# B&R Automation Studio project Cognex_V1_5
Automation Studio 4.6.3.55

## Configuration PP500_15

CPU , AutomationRuntime B4.62, Build 4.1.2, Safety 1.6, Vc V4.62.0

### Task classes (Cpu.sw)
```
Cyclic#8 (cycle 4000 us):
  Cognex <- Cognex.prg
  CognexVisN <- CognexVisNativeMode.prg
  CognexVisC <- CognexVisCommissioning.prg
  CognexVisA <- CognexVisArchive.prg
  CognexVisM <- CognexVisMain.prg
VcDataObjects: Visu <- Visu.dob, Visu1 <- Visu.dob
Binaries: vcclbox, vcctext, vcrt, vcresman, vccbar, vccstr, vccurl, vcchtml, vcpfmtcx, vcptelo, vcfile, vcdsint, vcpdsw, vccshape, arial, vccbmp, vcmgr, vcpdi855, vcshared, Visu01, vcdsloc, vcfntttf, vccovl, vctcal, arialbd, vcalarm, vcpfpp50, vccnum, vccline, vcpdi815, vccbtn, vcgclass, vcbclass, vcxml, Visu02, Visu03, visvc, vcpdvnc, vcnet, arconfig, sysconf, ashwd, asfw, iomap, vccalarm
Libraries: asieccon, asstring, astime, runtime, FileIO, Visapi, standard, BR_ATL_BMP, BR_ATL_LOG, sys_lib, dataobj, BR_ATL_COG, AsTCP, ethernet, AsICMP
```

### Hardware
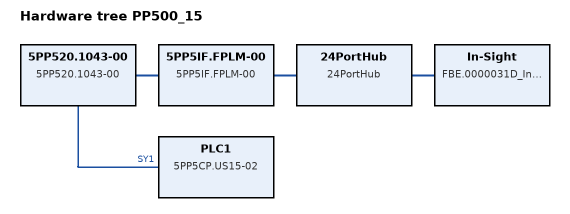
```
24PortHub : 24PortHub v1.0.0.1  [ETH1 -> 5PP5IF.FPLM-00.IF1 [Cable Type=PowerlinkCable, Length=10, Version=1.0.0.2]; ETH2 -> In-Sight.PLK1 [Cable Type=PowerlinkCable, Length=10, Version=1.0.0.2]]
5PP520.1043-00 : 5PP520.1043-00 v2.0.3.1
  Connector IF3:
    ActivateDevice = 1
    Mode = Manual
    SubnetMask = 255.255.0.0
    Vnc1
    VncVcObjectName1 = Visu
    VncAuthentication1 = 1
    VncPasswordViewOnly1 = r
    VncPasswordViewControl1 = w
  VcObjectName = Visu1
5PP5IF.FPLM-00 : 5PP5IF.FPLM-00 v2.4.0.0  [SL -> 5PP520.1043-00.SL1]
  Connector IF1:
    MtuSize = 1500
    CycleTime = 400
    InternetAddress = 10.16.7.34
    SubnetMask = 255.255.0.0
In-Sight : FBE.0000031D_In-Sight-7000 v4.7.1 (OrderNumber=In-Sight)  [PLK1 -> 24PortHub.ETH2 (NodeNumber=1) [Cable Type=PowerlinkCable, Length=10, Version=1.0.0.2]]
  Supervision = off
  p2000s01_direction = wo
  p2000s02_direction = wo
  p2001s01_direction = ro
  p2001s02_direction = ro
  p2010s01_direction = ro
  p2011s01_direction = ro
  p2011s02_direction = ro
  p2011s03_direction = ro
  p2011s04_direction = ro
  p2011s05_direction = ro
  p2011s06_direction = ro
  p2011s07_direction = ro
  p2011s08_direction = ro
  p2011s09_direction = ro
  p2011s0A_direction = ro
  p2011s0B_direction = ro
  p2021s01_direction = wo
  p2021s02_direction = wo
  p2021s03_direction = wo
PLC1 : 5PP5CP.US15-02 v2.0.6.0  [SY -> 5PP520.1043-00.SY1]
  PreserveNonVolatileSystemSettings = 0
  Connections = 8
  TimerDeviceType = EPLX2X
  TimerDevice = 5PP5IF.FPLM-00.IF1
  TaskClassIdleTime = 800
  Cyclic1Duration = 2000
  Cyclic1Tolerance = 2000
  Cyclic1Stack = 65535
  Cyclic2Stack = 65535
  Cyclic3Stack = 65535
  Cyclic4Stack = 65535
  Cyclic5Stack = 65535
  Cyclic6Stack = 65535
  Cyclic7Stack = 65535
  Cyclic8Duration = 4000
  Cyclic8Stack = 65535
```

### IoMap.iom - PLC1/IoMap.iom
```iecst
(********************************************************************
 * COPYRIGHT --
 ********************************************************************
 * File: IoMap.iom
 * Author: strickers
 * Created: May 16, 2012
 ********************************************************************
 * IO mapping file
 ********************************************************************)
VAR_CONFIG
	Cognex:cognex1sta AT %ID."In-Sight".Status_I2001_S01;
	Cognex:cognex1cmd AT %QD."In-Sight".Control_I2000_S01;
	cognex_1.sta.connected_plk AT %IX."In-Sight".ModuleOk;
	Cognex:tmpBarcodeRead1 AT %ID."In-Sight".InspectionResults_I2011_S01;
	Cognex:tmpBarcodeRead2 AT %ID."In-Sight".InspectionResults_I2011_S02;
	Cognex:tmpBarcodeRead3 AT %ID."In-Sight".InspectionResults_I2011_S03;
	Cognex:tmpBarcodeWrite1 AT %QD."In-Sight".UserData_I2021_S01;
	Cognex:tmpBarcodeWrite2 AT %QD."In-Sight".UserData_I2021_S02;
	Cognex:tmpBarcodeWrite3 AT %QD."In-Sight".UserData_I2021_S03;
	Cognex:tmpTextRead1 AT %ID."In-Sight".InspectionResults_I2011_S04;
	Cognex:tmpTextRead2 AT %ID."In-Sight".InspectionResults_I2011_S05;
	Cognex:tmpTextRead3 AT %ID."In-Sight".InspectionResults_I2011_S06;
	Cognex:tmpData1 AT %ID."In-Sight".InspectionResults_I2011_S07;
	Cognex:tmpData2 AT %ID."In-Sight".InspectionResults_I2011_S08;
	Cognex:tmpData3 AT %ID."In-Sight".InspectionResults_I2011_S09;
	Cognex:tmpData4 AT %ID."In-Sight".InspectionResults_I2011_S0A;
	cognex_1.cmd.job_id AT %QW."In-Sight".JobLoadID_I2000_S02;
	cognex_1.sta.job_id AT %IW."In-Sight".CurrentJobID_I2001_S02;
	Cognex:tmpData5 AT %ID."In-Sight".InspectionResults_I2011_S0B;
END_VAR
```

## Logical view

Binary libraries used (declarations not repeated): BR_ATL_LOG, sys_lib, Visapi

- 3_Powerlink.job (binary file, 1209220 bytes)
### Cognex.var
```iecst
(*-------------------------------------------------------------------------------------------------------------------------------------------------------------------------------------------------------------------------*)
VAR
	cognex1cmd : UDINT;
	cognex1sta : UDINT;
END_VAR
(*-------------------------------------------------------------------------------------------------------------------------------------------------------------------------------------------------------------------------*)
VAR
	strBarcodeWrite : STRING[20];
	strBarcodeWriteOld : STRING[20];
	strBarcodeRead : STRING[20];
	tmpBarcodeRead1 : UDINT;
	tmpBarcodeRead2 : UDINT;
	tmpBarcodeRead3 : UDINT;
	tmpBarcodeWrite1 : UDINT;
	tmpBarcodeWrite2 : UDINT;
	tmpBarcodeWrite3 : UDINT;
	BarcodeFixtureAngle : REAL;
	BarcodePass : USINT;
END_VAR
(*-------------------------------------------------------------------------------------------------------------------------------------------------------------------------------------------------------------------------*)
VAR
	strTextRead : STRING[20];
	TextExecutionTime : REAL;
	tmpTextRead1 : UDINT;
	tmpTextRead2 : UDINT;
	tmpTextRead3 : UDINT;
END_VAR
(*-------------------------------------------------------------------------------------------------------------------------------------------------------------------------------------------------------------------------*)
VAR
	tmpData1 : UDINT;
	tmpData2 : UDINT;
	tmpData3 : UDINT;
	tmpData4 : UDINT;
	tmpData5 : UDINT;
	tmp_inspecting_complete : BOOL;
	tmp_job_complete : BOOL;
	JobPass : USINT;
	JobExecutionTime : REAL;
	ComparePass : USINT;
	TextPass : USINT;
	FixturePass : USINT;
	ICMPping_0 : IcmpPing;
END_VAR
```

### Program Logical/CognexVisArchive

#### CognexVisArchive.ab
```automation-basic
(********************************************************************
 * COPYRIGHT --
 ********************************************************************
 * Author: strickers
 * Version: 1.0
 * This task has the following purpose
 * - Maintain a logbook with events coming from the camera
 * - Check the directory \Cognex for new pictures from the camera
 * - Convert the pictures from 8 Bit to 24 Bit so that they can be
 *   displayed in Visual Components
 * - Limit the amount of pictures and delete old if necessary
 * - Show picture archive and display old pictures
 * - Handle basic VC tasks like show/hide objects etc.
 ********************************************************************)

PROGRAM _INIT
	(* --------------------------------------------------------------------------------------------------------- *)
	(* Create file device for Cognex files and configuration files *)
	LOOP
		DevLink_0.enable 	= 1
		DevLink_0.pDevice 	= ADR("root")
		DevLink_0.pParam 	= ADR("/DEVICE=C:\\")
		DevLink_0 FUB DevLink()
		EXITIF(DevLink_0.status <> 65535)
	ENDLOOP
	(* --------------------------------------------------------------------------------------------------------- *)
	(* Create cognex folder for bitmaps on boot up *)
	LOOP
		DirCreate_0.enable 	= 1
		DirCreate_0.pDevice = ADR("root")
		DirCreate_0.pName 	= ADR("cognex_pics")
		DirCreate_0 FUB DirCreate()
		EXITIF(DirCreate_0.status <> 65535)
	ENDLOOP
	(* --------------------------------------------------------------------------------------------------------- *)
	(* Create file device for Cognex files and configuration files *)
	LOOP
		DevLink_0.enable 	= 1
		DevLink_0.pDevice 	= ADR("CognexPictures")
		DevLink_0.pParam 	= ADR("/DEVICE=C:\\cognex_pics")
		DevLink_0 FUB DevLink()
		EXITIF(DevLink_0.status <> 65535)
	ENDLOOP
	(* --------------------------------------------------------------------------------------------------------- *)
	VChandle = VA_Setup(1, "Visu")
	dir_entry_max =  SIZEOF(dir_data)/SIZEOF(dir_data[0])-1
END_PROGRAM

PROGRAM _CYCLIC
	(* --------------------------------------------------------------------------------------------------------- *)
	(* Display camera pictures from archieve *)
	(* --------------------------------------------------------------------------------------------------------- *)
	CASE step_diag OF
		(* --------------------------------------------------------------------------------------------------------- *)
		ACTION STP_INIT:
			(* Limit selection to last file name *)
			IF((dir_name_selected <> dir_name_selected_old) AND (dir_name_selected >= dir_name_selected_max) AND (dir_name_selected_max > 0)) THEN
				dir_name_selected		= dir_name_selected_max-1
				dir_name_selected_old 	= dir_name_selected
			(* Refresh file name list *)
			ELSE IF (vkDirRefresh) THEN
				memset(ADR(dir_names), 0, SIZEOF(dir_names))
				dir_name_selected_max = 0
				dir_entry = 0
				step_diag = STP_DIR_READ
			(* Display new selected picture *)
			ELSE IF (dir_name_selected <> dir_name_selected_old) THEN
				dir_name_selected_old = dir_name_selected
				VCbitmap_tmp = 0
				step_diag = STP_VC_LOAD
			ENDIF
		ENDACTION
		(* --------------------------------------------------------------------------------------------------------- *)
		ACTION STP_DIR_READ:
			(* Read all file names and date stamps from directory *)
			DirRead_0.enable 	= 1
			DirRead_0.pDevice 	= ADR("CognexPictures")
			DirRead_0.entry 	= dir_entry
			DirRead_0.option 	= fiFILE
			DirRead_0.pData 	= ADR(dir_data[dir_entry])
			DirRead_0.data_len 	= SIZEOF(dir_data[dir_entry])
			DirRead_0 FUB DirRead()
			(* Stop reading files when max number is reached *)
			IF (DirRead_0.status = fiERR_NO_MORE_ENTRIES) OR ((DirRead_0.status = 0) AND (dir_entry = dir_entry_max)) THEN
				step_diag = STP_DIR_EVAL
			(* Its all good, read next entry *)
			ELSE IF (DirRead_0.status = 0) THEN
				dir_entry = dir_entry + 1
				step_diag = STP_DIR_READ
			(* Jump to error step when FB faults *)
			ELSE IF (DirRead_0.status <> 65535) THEN
				NewLogEntry("#Error: dir read", ADR(logbook), 20)
				step_diag = STP_ERROR
			ENDIF
		ENDACTION
		(* --------------------------------------------------------------------------------------------------------- *)
		ACTION STP_DIR_EVAL:
			IF (dir_entry <> 0) THEN
				(* Extract file names from structure *)
				LOOP x=0 TO dir_entry-1 DO
					IF(memcmp(ADR(dir_data[x].Filename), ADR("cbrplc"), 6) = 0) THEN
						strcpy(ADR(dir_names[dir_name_selected_max]), ADR(dir_data[x].Filename[0]))
						dir_name_selected_max = dir_name_selected_max + 1
					ENDIF
				ENDLOOP
				(* Load first picture in list *)
				dir_name_selected 	= 0
				VCbitmap_tmp 		= 0
				step_diag 			= STP_VC_LOAD
			ELSE
				step_diag = STP_INIT
			ENDIF
			vkDirRefresh = 0
		ENDACTION
		(* --------------------------------------------------------------------------------------------------------- *)
		ACTION STP_VC_LOAD:
			(* Load picture into memory *)
			IF(VA_Saccess(1, VChandle) = 0) THEN
				VCerror = VA_LoadBitmap(1, VChandle, "CognexPictures", dir_names[dir_name_selected], ADR(VCbitmap_tmp))
				IF(VCerror = 0) THEN
					VCbitmap ACCESS VCbitmap_tmp
					step_diag = STP_VC_SHOW
				ELSE IF (VCerror <> 7000) THEN
					NewLogEntry("#Error: load bitmap", ADR(logbook), 20)
					step_diag = STP_ERROR
				ENDIF
				VA_Srelease(1, VChandle)
			ENDIF
		ENDACTION
		(* --------------------------------------------------------------------------------------------------------- *)
		ACTION STP_VC_SHOW:
			(* Display new picture *)
			IF(VA_Saccess(1, VChandle) = 0) THEN
				VCerror = VA_BlitBitmap(1, VChandle, ADR(VCbitmap), 700, 145, 700, 145, 700+PictureWidth, 145+PictureHeight, 1)
				IF(VCerror = 0) THEN
					VCbitmap ACCESS VCbitmap_tmp
					step_diag = STP_VC_FREE
				ELSE IF (VCerror <> 7000) THEN
					NewLogEntry("#Error: show bitmap", ADR(logbook), 20)
					step_diag = STP_ERROR
				ENDIF
				VA_Srelease(1, VChandle)
			ENDIF
		ENDACTION
		(* --------------------------------------------------------------------------------------------------------- *)
		ACTION STP_VC_FREE:
			(* Free up memory *)
			IF(VA_Saccess(1, VChandle) = 0) THEN
				VCerror = VA_FreeBitmap(1, VChandle, ADR(VCbitmap))
				IF(VCerror = 0) THEN
					VCbitmap ACCESS VCbitmap_tmp
					step_diag = STP_INIT
				ELSE IF (VCerror <> 7000) THEN
					NewLogEntry("#Error: free bitmap", ADR(logbook), 20)
					step_diag = STP_ERROR
				ENDIF
				VA_Srelease(1, VChandle)
			ENDIF
		ENDACTION
		(* --------------------------------------------------------------------------------------------------------- *)
		ACTION STP_ERROR:

		ENDACTION
	ENDCASE
END_PROGRAM
```

- Program Logical/CognexVisCommissioning (IEC) (no source held here)

- Program Logical/CognexVisNativeMode (IEC) (no source held here)

### Library Logical/Libraries/BR_ATL_BMP (ANSIC)
Depends on: FileIO

#### BR_ATL_BMP.fun - Exported functions and function blocks
```iecst
(********************************************************************
 * COPYRIGHT --
 ********************************************************************
 * Library: BR_ATL_BMP
 * File: BR_ATL_BMP.fun
 * Author: strickers
 * Created: May 23, 2012
 ********************************************************************
 * Functions and function blocks of library BR_ATL_BMP
 ********************************************************************)

FUNCTION_BLOCK BmpConvert
	VAR_INPUT
		enable : USINT;
		pDevice : UDINT;
		pFileSource : UDINT;
		pFileDestination : UDINT;
	END_VAR
	VAR_OUTPUT
		status : UINT;
	END_VAR
	VAR
		internal : typ_bmp_internal;
	END_VAR
END_FUNCTION_BLOCK
```

#### BR_ATL_BMP_LOC.h
```c
/********************************************************************
 * COPYRIGHT --
 ********************************************************************
 * Library: BR_ATL_BMP
 * File: BR_ATL_loc.h
 * Author: strickers
 * Created: May 23, 2012
 *******************************************************************/

#include <bur/plctypes.h>
#include <AsString.h>
#include <string.h>
#include <sys_lib.h>
#include <fileio.h>

/************************************************************************************************/
/*	Constants definition																		*/
/************************************************************************************************/
/* Constants for main step																		*/
#define STP_INIT			0
#define STP_SRC_OPEN		10
#define STP_SRC_READ		20
#define STP_SRC_CLOSE		30
#define STP_SRC_EVAL		40
#define STP_SRC_CONVERT		50
#define STP_DST_DELETE		60
#define STP_DST_CREATE		70
#define STP_DST_WRITE		80
#define STP_DST_CLOSE		90

#define STP_ERROR			100

#define BUSY				65535		/* Constant for status BUSY								*/
#define NO_ENABLE			65534
#define OK					0			/* Constant for status OK								*/

#define ERR_NO_DEVICE		10000
#define ERR_NO_SOURCE		10001
#define ERR_NO_DESTINATION	10002
#define ERR_NO_BMP_FILE		20000
#define ERR_FILE_TOO_BIG	20001
#define ERR_NOT_8BIT		20002

#define MAX_FILE_SIZE		100000
#define PIXEL_PER_CYCLE		1000

USINT in_buffer[MAX_FILE_SIZE];
USINT out_buffer[MAX_FILE_SIZE*3];

/************************************************************************************************/
/*	Version																						*/
/************************************************************************************************/
/* 1.0 First release																			*/
```

Listed in the project but not available here: Logical/CognexVisCommissioning/CognexVisCommissioning.ab, Logical/CognexVisCommissioning/CognexVisCommissioning.typ, Logical/CognexVisCommissioning/CognexVisCommissioning.var, Logical/CognexVisNativeMode/CognexVisNativeMode.ab, Logical/CognexVisNativeMode/CognexVisNativeMode.typ, Logical/CognexVisNativeMode/CognexVisNativeMode.var, Logical/Libraries/BR_ATL_BMP/BR_ATL_BMP.typ, Logical/Libraries/BR_ATL_BMP/BR_ATL_BMP.var, Logical/Libraries/BR_ATL_BMP/BR_ATL_BMP.c
